// TIA Portal V15.1 export
// export: Created 2020-06-12T07:35:54.6162109Z, ExportSetting None, DisplayName Totally Integrated Automation Portal, DisplayVersion V15.1, DisplayName TIA Portal Openness, DisplayVersion V15.1, DisplayName STEP 7 Professional, DisplayVersion V15.1, DisplayName STEP 7 Safety, DisplayVersion V15.1, DisplayName WinCC Advanced, DisplayVersion V15.1
FUNCTION "Signals_call" : Void   // FC1213, FBD
TITLE = General Program
{ S7_Optimized_Access := 'FALSE' }
// stored: AutoNumber false, SetENOAutomatically False
   VAR_TEMP
      _slag_bin_press : Bool;
      tAlarmSig : Bool;
      tAlarm : Bool;
      tAlarmDisable : Bool;
      tAlarmOn : Bool;
      tMeltAlarm : Bool;
      tCWAlarm : Bool;
   END_VAR
   VAR_TEMP   // added for the SCL form of the ladder/FBD networks
      _w1 : Bool;
      _w2 : Bool;
   END_VAR
BEGIN

REGION Network 1: ES1GM01 Lamp: Electrode Carriage Brake Locked
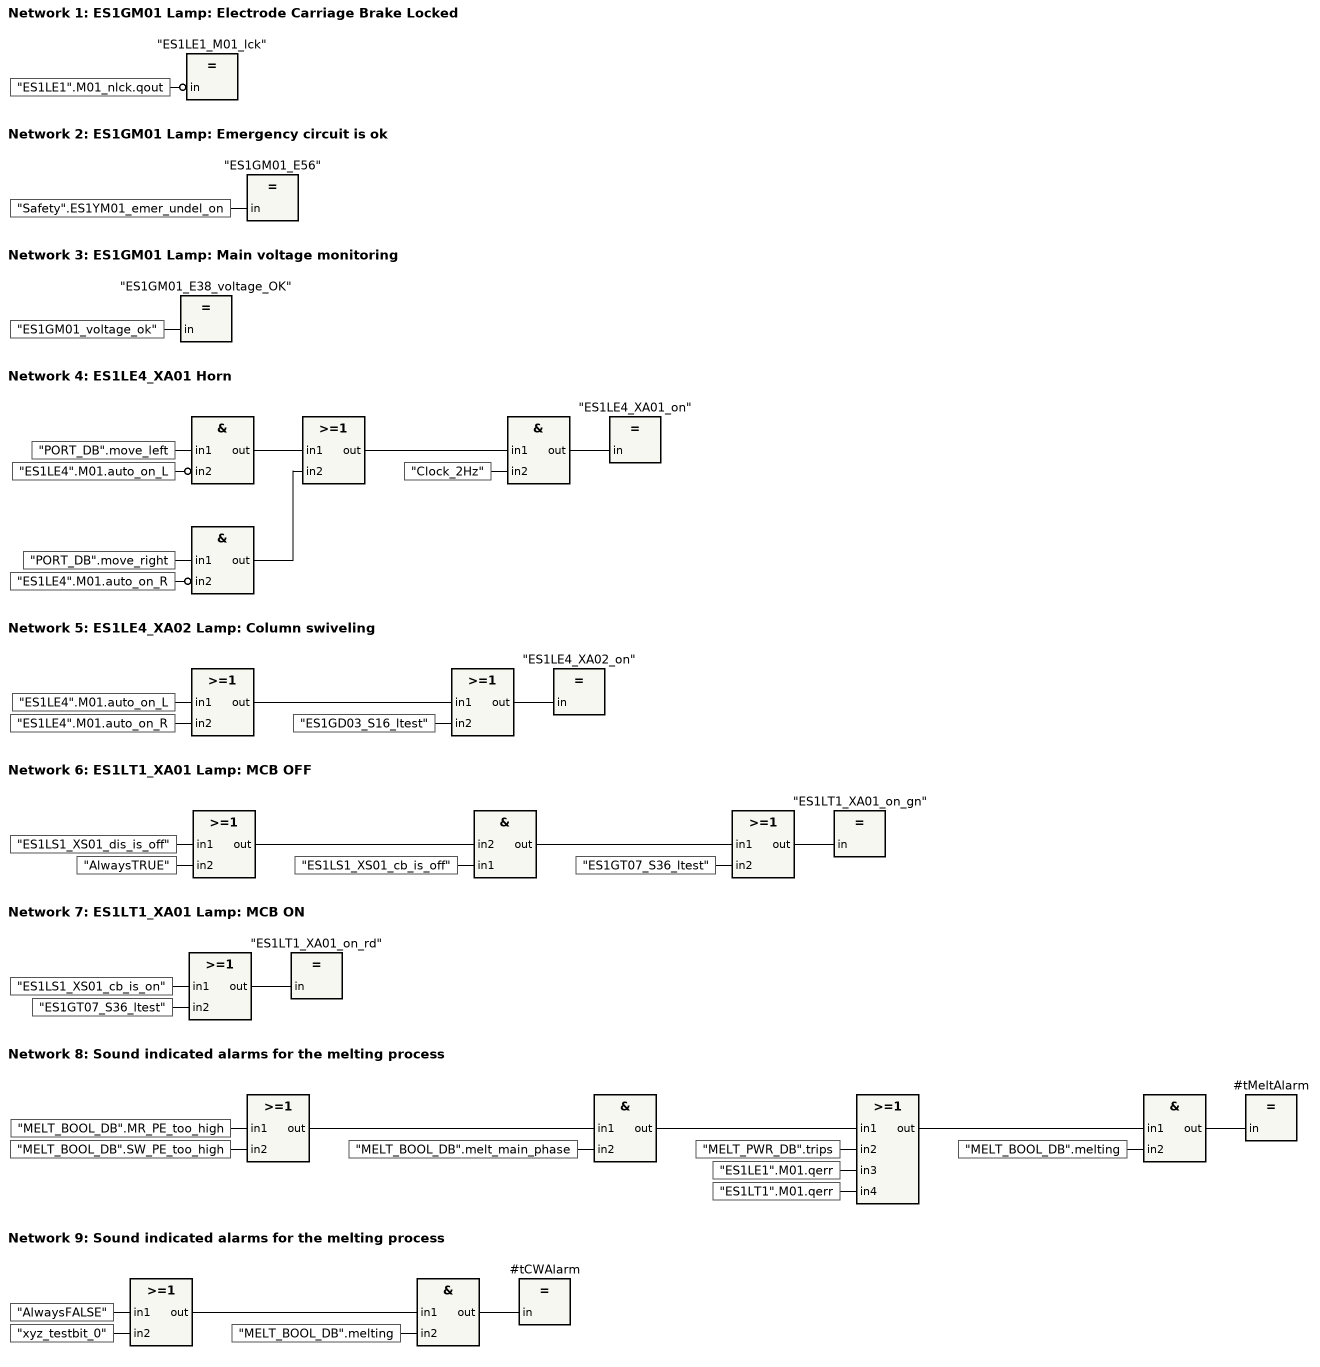
   "ES1LE1_M01_lck" := NOT "ES1LE1".M01_nlck.qout;
END_REGION

REGION Network 2: ES1GM01 Lamp: Emergency circuit is ok
   "ES1GM01_E56" := "Safety".ES1YM01_emer_undel_on;
END_REGION

REGION Network 3: ES1GM01 Lamp: Main voltage monitoring
   "ES1GM01_E38_voltage_OK" := "ES1GM01_voltage_ok";
END_REGION

REGION Network 4: ES1LE4_XA01 Horn
   "ES1LE4_XA01_on" := (("PORT_DB".move_left AND NOT "ES1LE4".M01.auto_on_L) OR ("PORT_DB".move_right AND NOT "ES1LE4".M01.auto_on_R)) AND "Clock_2Hz";
END_REGION

REGION Network 5: ES1LE4_XA02 Lamp: Column swiveling
   "ES1LE4_XA02_on" := "ES1LE4".M01.auto_on_L OR "ES1LE4".M01.auto_on_R OR "ES1GD03_S16_ltest";
END_REGION

REGION Network 6: ES1LT1_XA01 Lamp: MCB OFF
   // Delete me later:
   // "ES1LT1_XA01_on_gn"
   "ES1LT1_XA01_on_gn" := (("ES1LS1_XS01_dis_is_off" OR "AlwaysTRUE") AND "ES1LS1_XS01_cb_is_off") OR "ES1GT07_S36_ltest";
END_REGION

REGION Network 7: ES1LT1_XA01 Lamp: MCB ON
   // Delete me later:
   // "ES1LT1_XA01_on_rd"
   "ES1LT1_XA01_on_rd" := "ES1LS1_XS01_cb_is_on" OR "ES1GT07_S36_ltest";
END_REGION

REGION Network 8: Sound indicated alarms for the melting process
   #tMeltAlarm := ((("MELT_BOOL_DB".MR_PE_too_high OR "MELT_BOOL_DB".SW_PE_too_high) AND "MELT_BOOL_DB".melt_main_phase) OR "MELT_PWR_DB".trips OR "ES1LE1".M01.qerr OR "ES1LT1".M01.qerr) AND "MELT_BOOL_DB".melting;
END_REGION

REGION Network 9: Sound indicated alarms for the melting process
   #tCWAlarm := ("AlwaysFALSE" OR "xyz_testbit_0") AND "MELT_BOOL_DB".melting;
END_REGION

REGION Network 10: Collect important alarms
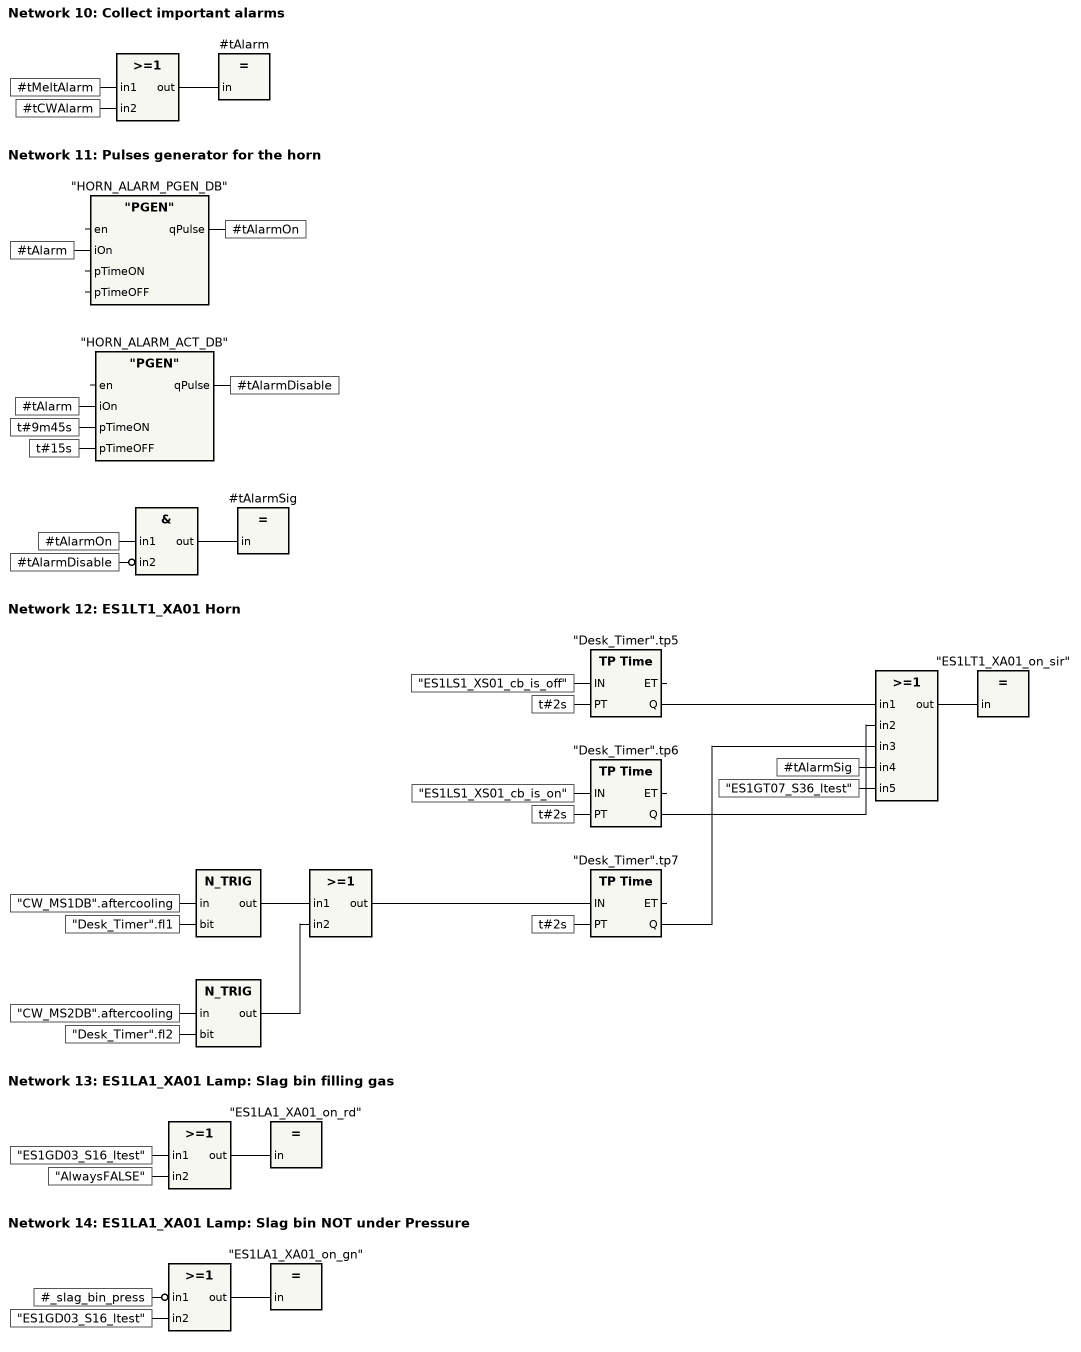
   #tAlarm := #tMeltAlarm OR #tCWAlarm;
END_REGION

REGION Network 11: Pulses generator for the horn
   "HORN_ALARM_PGEN_DB"(iOn := #tAlarm, qPulse => #tAlarmOn);   // "PGEN"
   "HORN_ALARM_ACT_DB"(iOn := #tAlarm, pTimeON := t#9m45s, pTimeOFF := t#15s, qPulse => #tAlarmDisable);   // "PGEN"
   #tAlarmSig := #tAlarmOn AND NOT #tAlarmDisable;
END_REGION

REGION Network 12: ES1LT1_XA01 Horn
   // Delete me later:
   // "ES1LT1_XA01_on_sir"
   "Desk_Timer".tp5.TP(IN := "ES1LS1_XS01_cb_is_off", PT := t#2s);
   "Desk_Timer".tp6.TP(IN := "ES1LS1_XS01_cb_is_on", PT := t#2s);
   #_w1 := NOT "CW_MS1DB".aftercooling AND "Desk_Timer".fl1;   // falling edge
   "Desk_Timer".fl1 := "CW_MS1DB".aftercooling;
   #_w2 := NOT "CW_MS2DB".aftercooling AND "Desk_Timer".fl2;   // falling edge
   "Desk_Timer".fl2 := "CW_MS2DB".aftercooling;
   "Desk_Timer".tp7.TP(IN := #_w1 OR #_w2, PT := t#2s);
   "ES1LT1_XA01_on_sir" := "Desk_Timer".tp5.Q OR "Desk_Timer".tp6.Q OR "Desk_Timer".tp7.Q OR #tAlarmSig OR "ES1GT07_S36_ltest";
END_REGION

REGION Network 13: ES1LA1_XA01 Lamp: Slag bin filling gas
   // PT is absolut, overpressure >1100mBar
   "ES1LA1_XA01_on_rd" := "ES1GD03_S16_ltest" OR "AlwaysFALSE";
END_REGION

REGION Network 14: ES1LA1_XA01 Lamp: Slag bin NOT under Pressure
   "ES1LA1_XA01_on_gn" := NOT #_slag_bin_press OR "ES1GD03_S16_ltest";
END_REGION
END_FUNCTION
